ABB RobotStudio station: Yumi_PCSDK_test.rsstn

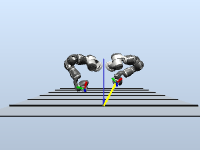
Station Yumi_PCSDK_test (saved by RobotStudio format 3)
Controller IRB_14000_0.5kg_0.5m, task T_ROB_L: task frame (RAPID world) sits at (0, 0, 0) mm, rotated rx 0 ry 0 rz 90 deg in the station
Controller IRB_14000_0.5kg_0.5m, task T_ROB_R: task frame (RAPID world) sits at (0, 0, 0) mm, rotated rx 0 ry 0 rz 90 deg in the station
Controller IRB_14000_0.5kg_0.5m
  mechanical unit ROB_R: IRB14000_0.5_0.5_R, 6 joints, base frame (0, 1.73, 0) mm
  mechanical unit ROB_R_7: IRB14000_0.5_0.5_R, 1 joints, base frame (0, 1.73, 0) mm
  mechanical unit ROB_L: IRB14000_0.5_0.5_L, 6 joints, base frame (0, 1.73, 0) mm
  mechanical unit ROB_L_7: IRB14000_0.5_0.5_L, 1 joints, base frame (0, 1.73, 0) mm
Layout (positions relative to the parent item):
  - IRB14000_0.5_0.5_R [mechanism, from Robots\IRB14000_0.5_0.5_R.rslib] at (-1.73, 0, 0) mm, rotated rx 0 ry 0 rz 90 deg; joint values [1.1248, -0.7255, -1.7409, 0.4932, 2.3336, 1.0457, -0.9045] (rad or m)
  - IRB14000_0.5_0.5_L [mechanism, from Robots\IRB14000_0.5_0.5_L.rslib] at (-1.73, 0, 0) mm, rotated rx 0 ry 0 rz 90 deg; joint values [-0.5676, -1.6821, 2.5584, 1.0086, 4.8034, 1.172, 0.3818] (rad or m)
  - Frame_1 [frame]
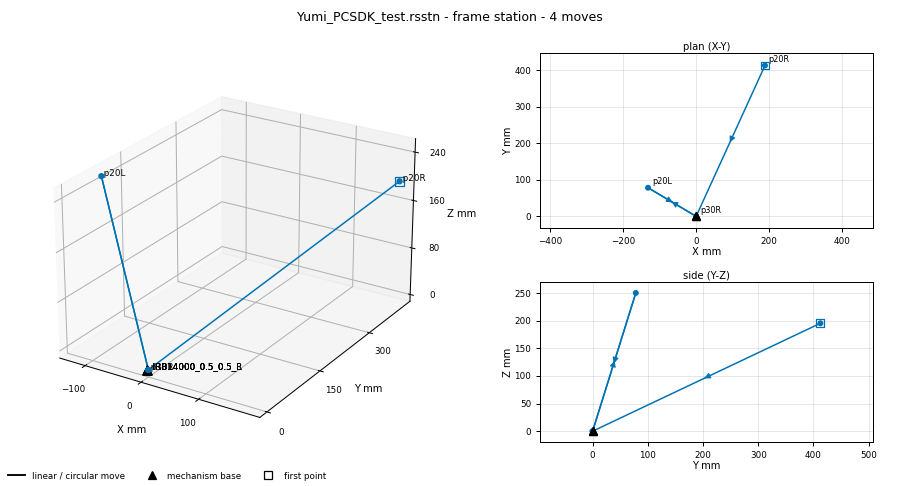
[picture p0: tool path of Yumi_PCSDK_test.rsstn in frame station, 4 of 4 moves have a stored position in this frame; points joined in program order, loops and branches not executed]
Targets, tools, work objects and paths stored in the station, written as RAPID:
! task T_ROB_R
MODULE MainModule
  VAR robtarget p20R:=[[412.53,-188.21,195.45],[0.0196523,0.791414,0.18309,0.582886],[0,1,-1,11],[150.954,9E9,9E9,9E9,9E9,9E9]];
  VAR robtarget p30R:=[[0,0,0],[1,0,0,0],[0,0,0,0],[9E9,9E9,9E9,9E9,9E9,9E9]];
  PROC main()
    ConfL \Off;
    MoveL p20R,v5000,z50,tool0;
    MoveL p30R,v5000,z50,tool0;
  ENDPROC
ENDMODULE

! task T_ROB_L
MODULE Module1
  PROC Path_10()
  ENDPROC
ENDMODULE

! task T_ROB_L
MODULE MainModule
  PERS robtarget p20L:=[[78.24,131.53,250.37],[0.167551944,0.793744733,0.389019869,0.436530853],[-1,3,0,11],[152.063,9E9,9E9,9E9,9E9,9E9]];
  VAR robtarget p30L:=[[0,0,0],[1,0,0,0],[0,0,0,0],[9E9,9E9,9E9,9E9,9E9,9E9]];
  TASK PERS wobjdata Workobject_1:=[FALSE,TRUE,"",[[0,0,0],[0,0,0,1]],[[0,0,0],[1,0,0,0]]];
  PROC main()
    ConfL \Off;
    MoveL p20L,v5000,z50,tool0\WObj:=wobj0;
    MoveL p30L,v5000,z50,tool0;
  ENDPROC
ENDMODULE

